FUNCTION_BLOCK FB_MachineControl EXTENDS FB_BaseTopElement
VAR

END_VAR

END_FUNCTION_BLOCK

(* stored: Version 1.1.0.1
   POU FB_MachineControl: Id {0eac6af2-3ab5-0548-0b1d-467819e04dee}, SpecialFunc None *)
